// TIA Portal project "START-RELEASE" (V16)

(* hardware
DEVICE "S7-1200 station_1"  S7-1200 Station
   slot 0: "Rack_0"  S7-1200 Rack  Rack  V1.0
   slot 1: "PLC_1"  CPU 1212C AC/DC/Rly  6ES7 212-1BE40-0XB0  V4.0
*)

// ===== PLC "PLC_1"  CPU 1212C AC/DC/Rly =====

VAR_GLOBAL   // PLC tag table "Default tag table"
   "START" AT %I0.2 : Bool;
   "STOP" AT %I0.3 : Bool;
   "KM1" AT %Q0.0 : Bool;
   "KM2" AT %Q0.1 : Bool;
   "KM3" AT %Q0.2 : Bool;
   "KM4" AT %Q0.3 : Bool;
   "LOOP MARKER" AT %M0.0 : Bool;
   "Tag_1" AT %M0.1 : Bool;
   "KM2 SS" AT %M0.2 : Bool;
   "KM3 SS" AT %M0.3 : Bool;
   "Tag_2" AT %M0.4 : Bool;
END_VAR

// folder: System blocks/Program resources

DATA_BLOCK "T1"   // DB1
{ S7_Optimized_Access := 'TRUE' }
AUTHOR : Simatic
FAMILY : IEC
NAME : IEC_TMR
VERSION : 1.0
// stored: InstanceOfName IEC_TIMER
"IEC_TIMER"
BEGIN
END_DATA_BLOCK

DATA_BLOCK "T2"   // DB2
{ S7_Optimized_Access := 'TRUE' }
AUTHOR : Simatic
FAMILY : IEC
NAME : IEC_TMR
VERSION : 1.0
// stored: InstanceOfName IEC_TIMER
"IEC_TIMER"
BEGIN
END_DATA_BLOCK

DATA_BLOCK "C1"   // DB3
{ S7_Optimized_Access := 'TRUE' }
AUTHOR : Simatic
FAMILY : IEC
NAME : CNTR
VERSION : 1.0
// stored: InstanceOfName IEC_COUNTER
"IEC_COUNTER"
BEGIN
END_DATA_BLOCK

DATA_BLOCK "T3"   // DB4
{ S7_Optimized_Access := 'TRUE' }
AUTHOR : Simatic
FAMILY : IEC
NAME : IEC_TMR
VERSION : 1.0
// stored: InstanceOfName IEC_TIMER
"IEC_TIMER"
BEGIN
END_DATA_BLOCK

// folder: (top level)

ORGANIZATION_BLOCK "Main"   // OB1, LAD, ProgramCycle
TITLE = "Main Program Sweep (Cycle)"
{ S7_Optimized_Access := 'TRUE' }
VERSION : 0.1
   VAR_INPUT
      Initial_Call : Bool;   // Initial call of this OB
      Remanence : Bool;   // =True, if remanent data are available
   END_VAR
   VAR_TEMP   // added for the SCL form of the ladder/FBD networks
      _w1 : Bool;
   END_VAR
BEGIN

REGION Network 1
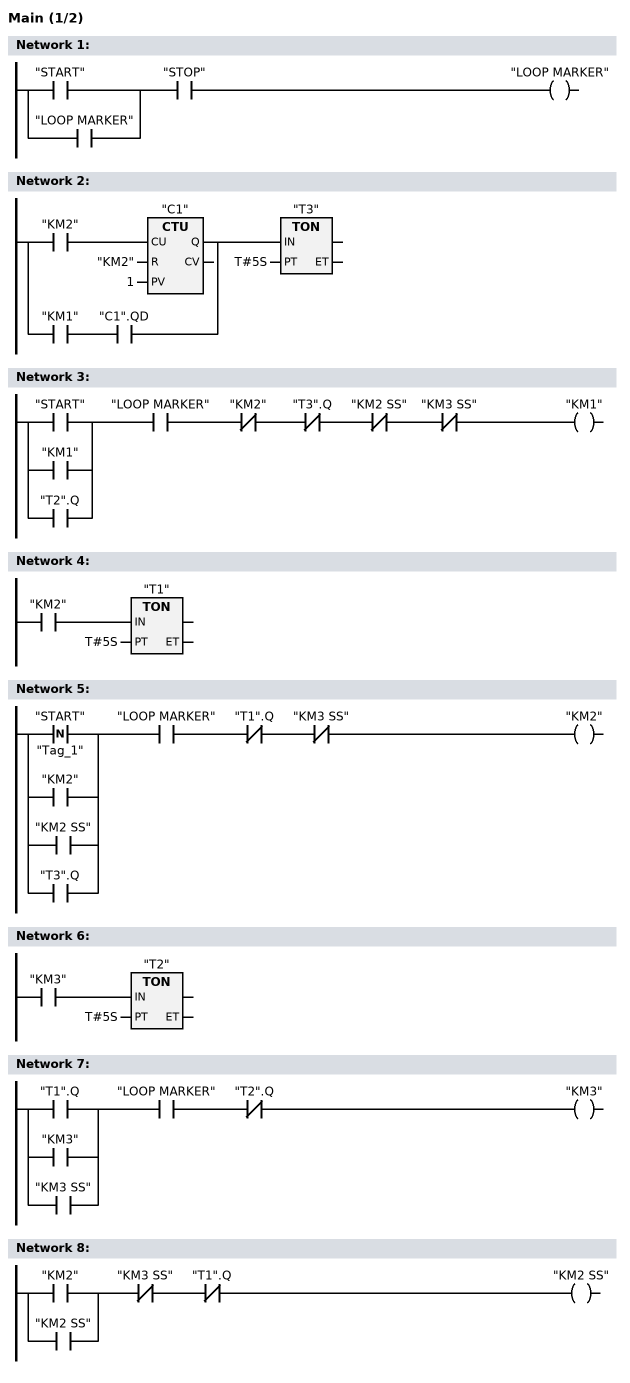
   RUNG wire#powerrail
      Contact( "START" )
      wire#w1
      Contact( "STOP" )
      Coil( "LOOP MARKER" )
   END_RUNG
   RUNG wire#powerrail
      Contact( "LOOP MARKER" )
   END_RUNG wire#w1
   // the same network as SCL:
   "LOOP MARKER" := ("START" OR "LOOP MARKER") AND "STOP";
END_REGION

REGION Network 2
   "C1".CTU(CU := "KM2", R := "KM2", PV := 1);
   "T3".TON(IN := "C1".Q OR ("KM1" AND "C1".QD), PT := T#5S);
END_REGION

REGION Network 3
   RUNG wire#powerrail
      Contact( "START" )
      wire#w1
      Contact( "LOOP MARKER" )
      I_Contact( "KM2" )
      I_Contact( "T3".Q )
      I_Contact( "KM2 SS" )
      I_Contact( "KM3 SS" )
      Coil( "KM1" )
   END_RUNG
   RUNG wire#powerrail
      Contact( "KM1" )
   END_RUNG wire#w1
   RUNG wire#powerrail
      Contact( "T2".Q )
   END_RUNG wire#w1
   // the same network as SCL:
   "KM1" := ("START" OR "KM1" OR "T2".Q) AND "LOOP MARKER" AND NOT "KM2" AND NOT "T3".Q AND NOT "KM2 SS" AND NOT "KM3 SS";
END_REGION

REGION Network 4
   "T1".TON(IN := "KM2", PT := T#5S);
END_REGION

REGION Network 5
   RUNG wire#powerrail
      N_Contact(operand := "START", bit := "Tag_1")
      wire#w1
      Contact( "LOOP MARKER" )
      I_Contact( "T1".Q )
      I_Contact( "KM3 SS" )
      Coil( "KM2" )
   END_RUNG
   RUNG wire#powerrail
      Contact( "KM2" )
   END_RUNG wire#w1
   RUNG wire#powerrail
      Contact( "KM2 SS" )
   END_RUNG wire#w1
   RUNG wire#powerrail
      Contact( "T3".Q )
   END_RUNG wire#w1
   // the same network as SCL:
   #_w1 := NOT "START" AND "Tag_1";   // falling edge of "START"
   "Tag_1" := "START";
   "KM2" := (#_w1 OR "KM2" OR "KM2 SS" OR "T3".Q) AND "LOOP MARKER" AND NOT "T1".Q AND NOT "KM3 SS";
END_REGION

REGION Network 6
   "T2".TON(IN := "KM3", PT := T#5S);
END_REGION

REGION Network 7
   RUNG wire#powerrail
      Contact( "T1".Q )
      wire#w1
      Contact( "LOOP MARKER" )
      I_Contact( "T2".Q )
      Coil( "KM3" )
   END_RUNG
   RUNG wire#powerrail
      Contact( "KM3" )
   END_RUNG wire#w1
   RUNG wire#powerrail
      Contact( "KM3 SS" )
   END_RUNG wire#w1
   // the same network as SCL:
   "KM3" := ("T1".Q OR "KM3" OR "KM3 SS") AND "LOOP MARKER" AND NOT "T2".Q;
END_REGION

REGION Network 8
   RUNG wire#powerrail
      Contact( "KM2" )
      wire#w1
      I_Contact( "KM3 SS" )
      I_Contact( "T1".Q )
      Coil( "KM2 SS" )
   END_RUNG
   RUNG wire#powerrail
      Contact( "KM2 SS" )
   END_RUNG wire#w1
   // the same network as SCL:
   "KM2 SS" := ("KM2" OR "KM2 SS") AND NOT "KM3 SS" AND NOT "T1".Q;
END_REGION

REGION Network 9
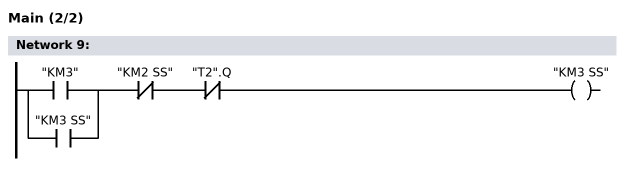
   RUNG wire#powerrail
      Contact( "KM3" )
      wire#w1
      I_Contact( "KM2 SS" )
      I_Contact( "T2".Q )
      Coil( "KM3 SS" )
   END_RUNG
   RUNG wire#powerrail
      Contact( "KM3 SS" )
   END_RUNG wire#w1
   // the same network as SCL:
   "KM3 SS" := ("KM3" OR "KM3 SS") AND NOT "KM2 SS" AND NOT "T2".Q;
END_REGION
END_ORGANIZATION_BLOCK